// TIA Portal V21 export
VAR_GLOBAL   // PLC tag table "K_NumAllarmi"
END_VAR
VAR_GLOBAL CONSTANT   // user constants
   K_NumAllarmiPerAnalogiche : Int := 5;
   K_NumAllarmiPerMotori : Int := 32;
   K_NumAllarmiPerZone : Int := 13;
   K_NumAllarmiPerValvole : Int := 4;
   K_NumAllarmiPerPid : Int := 3;
   K_NumAllarmiPerPortate : Int := 0;
   K_NumAllarmiPerParatie : Int := 3;
   K_NumAllarmiPerComunicazione : Int := 5;
   K_NumSlotAllarmiDaUtenze : Int := 5;
   K_NumAllarmiPerRicette : Int := 2;
   K_NumAllarmiPerSensori : Int := 1;
   K_NumAllarmiPerDispositivoProfinet : Int := 1;
   K_NumAllarmiPerSequenza : Int := 0;
   K_NumAllarmiPerSegnaliMacchina : Int := 3;
   K_NumAllarmiPerAdditivi : Int := 3;
END_VAR
